// TwinCAT 3 PLC project Untitled1
// ProgramVersion: 3.1.4024.0
// libraries:
//   Tc2_Standard, * (Beckhoff Automation GmbH)
//   Tc2_System, * (Beckhoff Automation GmbH)
//   Tc3_Module, * (Beckhoff Automation GmbH)
// project tree:
//   / GlobalTextList.TcGTLO, PlcTask.TcTTO, Visualization Manager.TcVMO (not stored)
//   GVLs/ GVL.TcGVL
//   POUs/ FB_EdgeDetector.TcPOU, F_A06.TcPOU, MAIN.TcPOU, averageCalculator.TcPOU, forgettingFactor.TcPOU, shiftLeft.TcPOU, PRG_DoSomeMath.TcPOU
//   VISUs/ Visualization.TcVIS
// real-time tasks:
//   TASK PlcTask: cycle T#10ms, priority 20, ADS port 350

CONFIGURATION Untitled1
    RESOURCE PLC ON TwinCAT3
        TASK PlcTask(INTERVAL := T#10ms, PRIORITY := 20);
        PROGRAM MAIN WITH PlcTask : MAIN;
    END_RESOURCE
END_CONFIGURATION

// ---- GVLs/GVL.TcGVL
{attribute 'qualified_only'}
VAR_GLOBAL
END_VAR

// ---- POUs/MAIN.TcPOU
PROGRAM MAIN
VAR
	//A4
	myWord : WORD := 16#5D7A;
	myWord2 : WORD;
	//A5
	myDWord : DWORD := 16#5D7A;
	myDWord2 : DWORD;
	myWord3 : WORD := 2#1111000011110000;
	
	//A7
	myRealArray: ARRAY[0..9] OF REAL := [1.1, 2.2, 3.3, 4.4, 5.5,6.6,7.7,8.8,9.9,10.10];  // Array mit 10 Elementen vom Typ REAL
	
	//A8
	index: INT;
	sum: REAL;
	mult: REAL;
	
	//A11
	bTasterblau : BOOL := TRUE;
	bTastergelb : BOOL := TRUE;
	blue_been_pressed : BOOL := FALSE;
	blue_led : BOOL := FALSE;
	blue_Counter : uint := 0;
	uiNumberPositiveEdgeBlue : UINT := 0;
	blueEdgeDetector : FB_EdgeDetector;
	yellowEdgeDetector : FB_EdgeDetector;
	
	//A13
	intUltrasonicSensor : INT;
	voltageUltrasonicSensor : REAL;
	
	//A14
	bufferArray : ARRAY[0..99] OF REAL ;
	
	
END_VAR

//frage wie kann man LED ansteueren?
//frage Ausgabe UltracSonic senosr?

//A4
myWord2 := SHR(myWord,3);
myDWord2 := SHL(myDWord,3);

//A5
myDWord2 := myWord OR 16#F0000000;

//A6
F_A06(16#1D06);

//A8
sum := 0;
mult := 1;
FOR index := 0 TO 9 DO
    sum := sum + myRealArray[index];  // Addiere den Schleifenindex zur Summe
	mult := mult * myRealArray[index];  // Addiere den Schleifenindex zur Summe
END_FOR;

//A9
sum := 0;
mult := 1;
index := 0;
WHILE index < 10 DO
	sum := sum + myRealArray[index];  // Addiere den Schleifenindex zur Summe
	mult := mult * myRealArray[index];  // Addiere den Schleifenindex zur Summe
	index := index +1;
END_WHILE;

//A10
index := 0;
REPEAT
    sum := sum + myRealArray[index];  // Addiere den Schleifenindex zur Summe
	mult := mult * myRealArray[index];  // Addiere den Schleifenindex zur Summe
	index := index +1;
UNTIL index < 10
END_REPEAT;

//A11
blueEdgeDetector(inputValue := bTasterblau, DoublePressedTime := 5);
IF blueEdgeDetector.risingEdge = TRUE THEN
	uiNumberPositiveEdgeBlue := uiNumberPositiveEdgeBlue + 1;
	
	//A12
	blue_been_pressed := NOT blue_been_pressed;
	blue_Counter := 0;
END_IF
yellowEdgeDetector(inputValue := bTastergelb, DoublePressedTime := 10);

//12
IF blue_been_pressed = TRUE THEN
	blue_Counter := blue_Counter + 1;
	IF blue_Counter >= 33 THEN
		blue_led := NOT blue_led;
		blue_Counter := 0;
	END_IF
END_IF

//A13
voltageUltrasonicSensor := intUltrasonicSensor / 10.0;

//A14
shiftLeft(bufferArray);
averageCalculator(bufferArray);

END_PROGRAM

// ---- POUs/FB_EdgeDetector.TcPOU
FUNCTION_BLOCK FB_EdgeDetector
VAR_INPUT
	inputValue : BOOL;
	DoublePressedTime: UINT;
END_VAR
VAR_OUTPUT
	risingEdge : BOOL;
	fallingEdge : BOOL;
	DoublePressed: BOOL;
END_VAR
VAR
	inputValue_old : BOOL;
	OncePressed: BOOL := FALSE;
	DoublePressedcounter: UINT := 0;
END_VAR

risingEdge := FALSE;
fallingEdge := FALSE;
DoublePressed := FALSE;

IF inputValue <> inputValue_old THEN
	IF inputValue = TRUE THEN
		risingEdge := TRUE;
		IF OncePressed = FALSE THEN
			OncePressed := TRUE;
		ELSE
			OncePressed := FALSE;
			DoublePressed := TRUE;
			DoublePressedcounter := 0;
		END_IF
	ELSE
		fallingEdge := TRUE;
	END_IF
END_IF
inputValue_old := inputValue;
IF OncePressed = TRUE THEN
	IF DoublePressedcounter >= DoublePressedTime THEN
		OncePressed := FALSE;
		DoublePressedcounter := 0;
	ELSE
		DoublePressedcounter := DoublePressedcounter + 1;
	END_IF	
END_IF

END_FUNCTION_BLOCK

// ---- POUs/F_A06.TcPOU


FUNCTION F_A06 : INT
VAR_INPUT
	rInput : WORD;
END_VAR
VAR
	inLenght : INT;
	overrunError: BOOL := FALSE;
	framingError: BOOL := FALSE;;
	parityError: BOOL := FALSE;;
	bufferFull: BOOL := FALSE;;
	initAccepted: BOOL := FALSE;;
	receiveRequest: BOOL := FALSE;;
	transmitAccepted: BOOL := FALSE;;
END_VAR

inLenght := WORD_TO_INT(SHR(rInput,8));
overrunError := WORD_TO_BOOL(rInput AND 16#40);
framingError := WORD_TO_BOOL(rInput AND 16#20);
parityError := WORD_TO_BOOL(rInput AND 16#10);
bufferFull := WORD_TO_BOOL(rInput AND 16#8);
initAccepted := WORD_TO_BOOL(rInput AND 16#4);
receiveRequest := WORD_TO_BOOL(rInput AND 16#2);
transmitAccepted := WORD_TO_BOOL(rInput AND 16#1);

RETURN;

END_FUNCTION

// ---- POUs/shiftLeft.TcPOU
FUNCTION shiftLeft : ARRAY[0..99] OF REAL
VAR_INPUT
	inputbuffer : ARRAY[0..99] OF REAL;
END_VAR
VAR
	tempIndex : UINT := 0;
	tempbuffer : ARRAY[0..99] OF REAL;
END_VAR

FOR tempIndex := 0 TO 98 DO
	tempbuffer[tempIndex] := inputbuffer[tempIndex+1];
END_FOR

shiftleft := tempbuffer;
RETURN;

END_FUNCTION

// ---- POUs/averageCalculator.TcPOU
FUNCTION averageCalculator : REAL
VAR_INPUT
	inputbuffer : ARRAY[0..99] OF REAL;
END_VAR
VAR
	tempIndex : INT := 0;
	tempSum :REAL := 0;
END_VAR

FOR tempIndex := 0 TO 99 DO
	tempSum := tempSum + inputbuffer[tempIndex];
END_FOR
averageCalculator := tempSum/100;
RETURN;

END_FUNCTION

// ---- POUs/forgettingFactor.TcPOU
FUNCTION_BLOCK forgettingFactor
VAR_INPUT
	inputValue : REAL;
END_VAR
VAR_OUTPUT
	meanValue : REAL;
END_VAR
VAR
	A_Factor : REAL := 0.5;
	y_um :REAL;
	meanValue_um : REAL;
END_VAR

meanValue := A_Factor * meanValue_um + (1-A_Factor)*y_um;

y_um := inputValue;
meanValue_um := meanValue;

END_FUNCTION_BLOCK

// ---- POUs/PRG_DoSomeMath.TcPOU
PROGRAM PRG_DoSomeMath
VAR_INPUT
	
END_VAR
VAR
	rVariable1 : REAL;
	rVariable2 : REAL;
	rVariable3 : REAL;
	rVariable4 : REAL;
	rPRG_Count : UINT;
END_VAR

rPRG_Count := rPRG_Count + 1;

rVariable1 := F_AdditionFunction(23.23,4.3);
rVariable2 := F_SubstractFunction(23.23,4.3);
rVariable3 := F_MultiplicationFunction(23.23,4.3);
rVariable4 := F_DivisionFunction(23.23,4.3);

END_PROGRAM

// ---- VISUs/Visualization.TcVIS
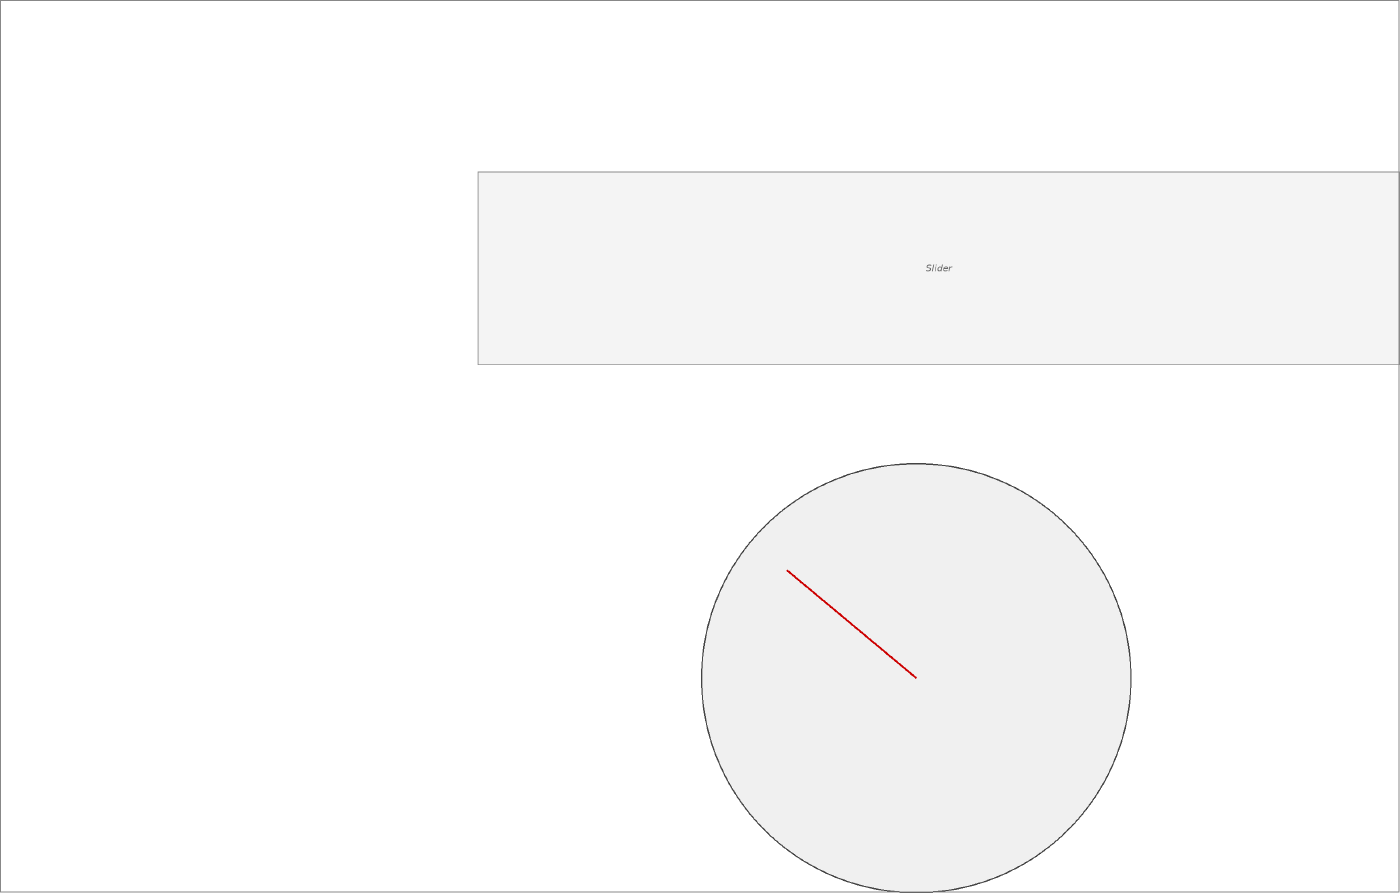
VISUALIZATION Visualization  // 1565x999
    Slider (534,192 1031x216), variable: MAIN.intUltrasonicSensor, scale 0..100
        p2541109501: MAIN.voltageUltrasonicSensor
    Meter180 (586,518 876x481), value: MAIN.voltageUltrasonicSensor, style: Meter-Meter180-Gray, scale format: %.1f, scale 0..10
END_VISUALIZATION
